VISUALIZATION Page_Main  // 1080x660, background image 
END_VISUALIZATION

(* stored: Version 1.1.0.1
   Visu Page_Main: Id {42215623-f4da-4207-8e8a-30a22be9faaa} *)
